FUNCTION_BLOCK INTERNAL FINAL ReceiverListExtender
VAR
	_iList		: I_ReceiverList;
END_VAR

PROPERTY INTERNAL List : I_ReceiverList
GET
List := _iList;
END_GET
SET
_iList := List;
END_SET
END_PROPERTY

END_FUNCTION_BLOCK

(* stored: Version 1.1.0.1
   POU ReceiverListExtender: Id {70918c97-6f50-4cac-862b-1465246836fd}, SpecialFunc None
   Property List: Id {f5b2f04a-332b-4755-9e45-aa4b076e8c53}
   Get Get: Id {e6958808-e26e-4000-a99e-1b29cd3e3059}
   Set Set: Id {83395991-4c47-4626-acb1-e3b3d9fa46df} *)
